PROGRAM MAIN
VAR
END_VAR


	PRG_Home();
	PRG_Testing();

END_PROGRAM

(* stored: Version 1.1.0.1, ProductVersion 3.1.4024.13
   POU MAIN: Id {d06f72d8-5174-4e47-9e6b-38c81cebdc5e}, SpecialFunc None *)
